TYPE "TExtEncoder_ErrorWord"
VERSION : 0.1
// Block: TExtEncoder_ErrorWord
   STRUCT
      SystemFault : Bool;
      ConfigFault : Bool;
      UserFault : Bool;
      CommandNotAccepted : Bool;
      SensorFault : Bool;
      CommunicationFault : Bool;
      HomingError : Bool;
      PeripheralError : Bool;
   END_STRUCT;

END_TYPE
